PROGRAM MAIN
VAR
	
END_VAR

P_ModbusMaster();
P_ModbusSlave();

END_PROGRAM

(* stored: Version 1.1.0.1, ProductVersion 3.1.4024.12
   POU MAIN: Id {d3daa20c-f2e3-400e-8eb6-142ce6db79be}, SpecialFunc None *)
